FUNCTION F_IsEmpty : BOOL
VAR_INPUT
	WX : sBogie;
END_VAR
VAR
END_VAR

IF WX.A.bPP1_Input = 0 AND WX.A.bPP2_Input = 0 AND WX.B.bPP2_Input = 0 AND WX.B.bPP2_Input = 0 THEN
	F_IsEmpty := 1;
	ELSE 
		F_IsEmpty := 0;
END_IF

END_FUNCTION

(* stored: Version 1.1.0.1, ProductVersion 3.1.4024.12
   POU F_IsEmpty: Id {ee171399-c061-4b46-88d9-82ec799cfc05}, SpecialFunc None *)
